PROGRAM System_Time
VAR
    fbLocalTime : FB_LocalSystemTime; (* FB 인스턴스 *)
    bEnable     : BOOL := TRUE;       (* FB 활성화 *)
    dwCycleTime : DWORD := 1;         (* 시간 동기화 주기 (1초) *)
    stCurrentTime : TIMESTRUCT;       (* 출력 시간 구조체 *)
    bValid      : BOOL;
    sTimeString : STRING;             (* 최종 출력 문자열 *)
	uliSystemTimeMs:  ULINT;
	F_GetCurTaskCycleTime: INT;
END_VAR


// PLC 사이클마다 실행됩니다.
//uliSystemTimeMs := F_GetSystemTime();

//GVL_System.Time_Data := uliSystemTimeMs;

END_PROGRAM

(* stored: Version 1.1.0.1, ProductVersion 3.1.4024.15
   POU System_Time: Id {c1745ddb-e23a-4e49-a256-e1b685177728}, SpecialFunc None *)
